// Process Simulation. All functionality packed into one method for easier overwriting
THIS^.Simulation();


// If enabled start station logic
IF THIS^.ipXtsSystem.Enabled THEN
	
	ipThisStation := (THIS^);
	//Detect mover who is passing the station whitout be in queue. Adjust to new Gap+Dynamics
	IF fbTrigger.MoverDetected AND fbTrigger.MoverAtTrigger<>0 AND NOT THIS^.bSuppressDynamicsChange THEN
		//Only if not in this queue
		IF fbTrigger.MoverAtTrigger.ParentStation <> ipThisStation THEN
			fbTrigger.MoverAtTrigger.MoveAbsCA(
				fPosition:= fbTrigger.MoverAtTrigger.LastCmdTargedPosition, 
				fVelocity:= THIS^.fMoverVelocityAtExit, 
				fGap:= THIS^.fMoverGapAtExit, 
				eDirection:= Tc3_Mc3Definitions.MC_DIRECTION.mcDirectionPositive);
		END_IF
	END_IF
	
	
	//Test if the first mover is in station and send him away, if the destination is not this station
	IF (THIS^.MoversInQueue[0] <> 0) AND_THEN (THIS^.MoversInQueue[0].TargedStation <> THIS^.StationGroupID) AND_THEN __QUERYINTERFACE(THIS^.MoversInQueue[0],ipMover) THEN
		//IF mover is standstill in current station, send him away whit the exitVelocity, else use the in mover stored velocity
		IF (THIS^.MoversInQueue[0].PositionOnTrack = THIS^.PositionOnTrack) THEN
			THIS^.TrySendMoverToNextStation(ipMover := ipMover, fVelocity := THIS^.fMoverVelocityAtExit, fGap := THIS^.fMoverGapAtExit);
		ELSE
			THIS^.TrySendMoverToNextStation(ipMover := ipMover, fVelocity := ipMover.LastCmdTargedVelocity, fGap := ipMover.LastCmdTargedGap);
		END_IF	
      
	END_IF
END_IF


// Utility InfoStation, used in XTS Viewer. All functionality packed into one method for easier overwriting
THIS^.UtilityStation();

// Calculate statistic values like Mover/min of this station. All functionality packed into one method for easier overwriting
THIS^.UpdateStatistic();
END_METHOD

METHOD PROTECTED UtilityStation : HRESULT //Utility InfoStation, used in XTS Viewer. All functionality packed into one method for easier overwriting
VAR
	aStopPositionsInfoStation : ARRAY[1..Tc3_XTS_Utility.TcIoXtsEnvironmentParameterList.MaxXtsStopPositionsPerStation] OF LREAL;
	fLastStopPosition 		: LREAL;
	nLoopIndex 				: UINT;	
    ipMovers 				: CHALET_BaseComponents.I_CH_List;
	ipTempMover 			: I_XTS_Mover;
	nXpuNo 					: UINT;
	nMoverNo 				: UINT;
END_VAR

VAR_INST
	bUtilityStationInitDone : BOOL;
	nOldMoverQueueSize 		: UINT := CHALET_BaseComponents.GVL_Datatypes.cMaxUint;
	fOldPositionOnTrack 	: LREAL;
	anBias 					: ARRAY[1..2] OF INT;
	bInverted 				: BOOL;
END_VAR
//Validate inputs
IF THIS^.OIDStationInfo = 0 OR ipXtsSystem.Environment = 0 THEN
	RETURN;
END_IF	


// Initalize
IF NOT bUtilityStationInitDone THEN
	//Get interface to utility station belongs to this station via OID
    FOR nLoopIndex := 1 TO ipXtsSystem.Environment.UtilityEnvirement.InfoServerTcIo(1).P_InfoStationCount DO
		IF 	ipXtsSystem.Environment.UtilityEnvirement.InfoServerTcIo(1).P_InfoStationOids[nLoopIndex] = THIS^.OIDStationInfo THEN
			THIS^.ipStationInfo := ipXtsSystem.Environment.UtilityEnvirement.InfoServerTcIo(1).InfoStationTcIo(nInfoStation:= nLoopIndex);
			EXIT;
		END_IF
	END_FOR	
	
	// calculate Position Offset
	IF THIS^.ipStationInfo <> 0 THEN			
		ipMovers := ipXtsSystem.Movers;
		ipMovers.ResetIterator();
		nLoopIndex := 0;	
		WHILE ipMovers.HasNextObject() DO
			nLoopIndex := nLoopIndex + 1;
			IF ToMover(ipMovers.GetNextObject(),ipTempMover) THEN
				//get Xpu Number by AxisId
				nXpuNo := ipXtsSystem.Environment.UtilityEnvirement.GetXpuNumberByAxisId(ipTempMover.getAxisRef.NcToPlc.AxisId);
				//get Mover Number by AxisId
				nMoverNo := ipXtsSystem.Environment.UtilityEnvirement.XpuTcIo(nXpuNo).GetMoverNumberByAxisId(ipTempMover.getAxisRef.NcToPlc.AxisId);
				//calculate Bias
				anBias[nLoopIndex] := LREAL_TO_INT(ipXtsSystem.Environment.UtilityEnvirement.XpuTcIo(nXpuNo).MoverTcIo(nMoverNo).GetPositionInfo().fPartPosition - ipTempMover.getAxisRef.NcToPlc.ModuloActPos);
				IF nLoopIndex = 2 THEN
					 EXIT;
				END_IF
			END_IF
		END_WHILE
		
		// Validate bias, check for inverted direction
		IF anBias[1] <> anBias[2] THEN
			bInverted := TRUE; 
			ipMovers.ResetIterator();
			nLoopIndex := 0;	
			WHILE ipMovers.HasNextObject() DO
				nLoopIndex := nLoopIndex + 1;
				IF ToMover(ipMovers.GetNextObject(),ipTempMover) THEN
					//get Xpu Number by AxisId
					nXpuNo := ipXtsSystem.Environment.UtilityEnvirement.GetXpuNumberByAxisId(ipTempMover.getAxisRef.NcToPlc.AxisId);
					//get Mover Number by AxisId
					nMoverNo := ipXtsSystem.Environment.UtilityEnvirement.XpuTcIo(nXpuNo).GetMoverNumberByAxisId(ipTempMover.getAxisRef.NcToPlc.AxisId);
					//calculate inverted Bias
					anBias[nLoopIndex] := LREAL_TO_INT(ipXtsSystem.TrackLength - ipXtsSystem.Environment.UtilityEnvirement.XpuTcIo(nXpuNo).MoverTcIo(nMoverNo).GetPositionInfo().fPartPosition - ipTempMover.getAxisRef.NcToPlc.ModuloActPos);
					IF nLoopIndex = 2 THEN
						 EXIT;
					END_IF
				END_IF	
			END_WHILE
		END_IF
		
		//Set unique station name
		THIS^.ipStationInfo.SetDescription(THIS^.LUID);

	END_IF
	bUtilityStationInitDone := TRUE;
END_IF




// Update
// Configure/draw station in viewer on change
IF (THIS^.ipStationInfo <> 0) AND (THIS^.nMoverQueueSize <> nOldMoverQueueSize OR THIS^.fPositionOnTrack <> fOldPositionOnTrack) THEN	
	nOldMoverQueueSize := THIS^.nMoverQueueSize;
	fOldPositionOnTrack := THIS^.fPositionOnTrack;
	
	
	
	// Draw stop position if gap between mover, given by station behind, is set
	IF (StationBehinde <> 0) AND (THIS^.nMoverQueueSize > 0) AND THIS^.nMoverQueueSize <= 25 THEN
		//Clear array
		MEMSET(ADR(aStopPositionsInfoStation), SIZEOF(aStopPositionsInfoStation), 0);
		//Fill array
		FOR nLoopIndex := 1 TO THIS^.nMoverQueueSize DO
			fLastStopPosition := (nLoopIndex-1)*StationBehinde.MoverGapAtExit;
			aStopPositionsInfoStation[(nLoopIndex)] := (fLastStopPosition);
		END_FOR
		IF NOT bInverted THEN
			//Start Position
			THIS^.ipStationInfo.SetStartPositionOnPart(MAX((fPositionOnTrack + anBias[1] - fLastStopPosition), 0)); ///zzz Todo. The InfoStation can not draw stations in the modulo area
			//End Pos
			THIS^.ipStationInfo.SetEndPositionOnPart(fPositionOnTrack + anBias[1]);
		ELSE
			//Start Position
			THIS^.ipStationInfo.SetStartPositionOnPart(ipXtsSystem.TrackLength - (fPositionOnTrack + anBias[1]));					
			//End Pos
			THIS^.ipStationInfo.SetEndPositionOnPart(MAX((ipXtsSystem.TrackLength - (fPositionOnTrack + anBias[1] - fLastStopPosition)), 0)); ///zzz Todo. The InfoStation can not draw stations in the modulo area
		END_IF
		//StopPositions
		THIS^.ipStationInfo.SetStopPositions(aStopPositionsInfoStation);

		//Override color if is set to transparent
		IF THIS^.ipStationInfo.GetStationColor() = 0 THEN
			THIS^.ipStationInfo.SetStationColor(nStationColor:= E_Colors_ARGB.Darkred);
		END_IF
	ELSE
		//Clear array
		MEMSET(ADR(aStopPositionsInfoStation), SIZEOF(aStopPositionsInfoStation), 0);	
		//StopPositions
		THIS^.ipStationInfo.SetStopPositions(aStopPositionsInfoStation);
		//Start Pos
		THIS^.ipStationInfo.SetStartPositionOnPart(nStartPositionOnPart := fPositionOnTrack + anBias[1]);
		//End Position
		THIS^.ipStationInfo.SetEndPositionOnPart(nEndPositionOnPart := fPositionOnTrack + anBias[1]);
	END_IF
	
	
	
	//Color Station depending on function:
	// Waitingstation green
	IF (FIND(THIS^.LUID,'wait')>0) OR (FIND(THIS^.LUID,'Wait')>0) OR (FIND(THIS^.LUID,'Warte')>0) OR (FIND(THIS^.LUID,'warte')>0) THEN
		THIS^.UtilityStationInfo.SetStationColor(nStationColor := E_Colors_ARGB.Green);
	
	// Dynamicstation blue
	ELSIF THIS^.MoverQueueSize = 0 THEN
		THIS^.UtilityStationInfo.SetStationColor(nStationColor := E_Colors_ARGB.Royalblue);	
    
	// Process station red
	ELSE
		THIS^.UtilityStationInfo.SetStationColor(nStationColor := E_Colors_ARGB.Red);			
	END_IF

END_IF
END_METHOD

{attribute 'monitoring':='call'}
PROPERTY UtilityStationInfo : I_TcIoXtsInfoServerInfoStation
GET
UtilityStationInfo := THIS^.ipStationInfo;
END_GET
END_PROPERTY

END_FUNCTION_BLOCK

// COMPENENTs/Trigger/FB_XTS_Trigger
{attribute 'no_explicit_call' := 'Do not call the body - Stick to OOP'}
FUNCTION_BLOCK FB_XTS_Trigger EXTENDS FB_CH_Object IMPLEMENTS I_XTS_Trigger
VAR
	{attribute 'hide'}
	bInitDone : BOOL;
	{attribute 'hide'}
	ipXtsSystem : I_XTS_System_Registration;
	{attribute 'hide'}
	ipListOfMoversToCheck : CHALET_BaseComponents.I_CH_LIST;
	{attribute 'hide'}
	fTriggerPositionOnTrack : LREAL;
	{attribute 'hide'}
	eTriggerDirection : Tc2_MC2.MC_Direction := MC_Positive_Direction;
	{attribute 'hide'}
	ipMoverAtTrigger : I_XTS_Mover;
	{attribute 'hide'}	
	fTrackLentgh : LREAL;
	{attribute 'hide'}
	aMoversPositionLastCycle : ARRAY [0..(XtsParameterlist.MAX_MOVER_PER_SYSTEM-1)] OF LREAL; // This list is generated at the end of the PRG and contais the positions. The positions are checked in the next cycle
	{attribute 'hide'}
	aMoversInterfaceLastCycle : ARRAY [0..(XtsParameterlist.MAX_MOVER_PER_SYSTEM-1)] OF I_XTS_Mover; // This list is generated at the end of the PRG and contais the Mover interface. The positions are checked in the next cycle
	
END_VAR

METHOD FB_init : BOOL
VAR_INPUT
	bInitRetains : BOOL; // if TRUE, the retain variables are initialized (warm start / cold start)
	bInCopyCode : BOOL;  // if TRUE, the instance afterwards gets moved into the copy code (online change)
	
	ipXtsSystem : I_XTS_System_Registration; //Interface to XTS system object
	
END_VAR
VAR_INST
	{attribute 'hide'}
	bFBInitCalledOnce : BOOL; //Do the following code once during start up and not during onlinechange
END_VAR
//Do the following code once during start up and not during onlinechange
IF NOT bFBInitCalledOnce THEN 
	;
END_IF

//Regristrate object in System if unknown
IF ipXtsSystem <> 0 AND THIS^.ipXtsSystem = 0 THEN
	ipXtsSystem.RegisterTrigger(THIS^);
	THIS^.ipXtsSystem := ipXtsSystem;
END_IF

bFBInitCalledOnce := TRUE;
END_METHOD

{attribute 'monitoring':='call'}
PROPERTY HR : HRESULT
GET
///zzz todo
END_GET
END_PROPERTY

METHOD Initialize : HRESULT
IF THIS^.ipXtsSystem = 0 THEN
	//No valide interface
	Initialize := E_FAIL;
	RETURN;
END_IF

//Store track information
THIS^.fTrackLentgh := THIS^.ipXtsSystem.TrackLength;

IF (THIS^.ipListOfMoversToCheck <> 0) AND (THIS^.fTrackLentgh > 0.0) THEN
	THIS^.bInitDone := TRUE;
	Initialize := S_OK;
ELSE
	Initialize := E_FAIL;
END_IF
END_METHOD

PROPERTY ListOfMoversToCheck : I_CH_List
SET
IF ListOfMoversToCheck <> 0 THEN
	ipListOfMoversToCheck := ListOfMoversToCheck;
END_IF
END_SET
END_PROPERTY

{attribute 'monitoring':='call'}
PROPERTY MoverAtTrigger : I_XTS_Mover
GET
THIS^.Prepare();//Prepare Time-critical information

MoverAtTrigger := ipMoverAtTrigger;
END_GET
END_PROPERTY

{attribute 'monitoring':='call'}
PROPERTY MoverDetected : BOOL
GET
THIS^.Prepare();//Prepare Time-critical information

MoverDetected := (ipMoverAtTrigger <> 0);
END_GET
END_PROPERTY

{attribute 'monitoring':='call'}
PROPERTY PositionOnTrack : LREAL
GET
PositionOnTrack := fTriggerPositionOnTrack;
END_GET
SET
fTriggerPositionOnTrack := PositionOnTrack;
END_SET
END_PROPERTY

(* Time-critical information is processed here, which can then be polled via the property every cycle. 
The update method is usually at the end of the program and then it is already 'outdated'. *)
METHOD PRIVATE Prepare : HRESULT
VAR
	fMoverActPos,fMoverLastPos : LREAL;
	fRangePositive, fRangeNegative : LREAL;
	bMoverWasInRangeNeg, bMoverWasInRangePos, bMoverIsInRangeNeg, bMoverIsInRangePos : BOOL;
	nLoopIndex : UINT;
END_VAR
VAR_INST
	{attribute 'hide'}
	nLastUpdatedCycleCount : UDINT;
END_VAR
VAR CONSTANT
	cMaxMoveDistPerCycle : LREAL := 4000.0 * 20.0 / 1000.0 * 1.1; //4 m/s(max. XTS speed) * 20ms(max realistic SPS cycle time) + 10%
END_VAR
//Check if this Cycle the dates are allready prepared
IF nLastUpdatedCycleCount <> TwinCAT_SystemInfoVarList._TaskInfo[THIS^.nTaskIndex].CycleCount THEN
	nLastUpdatedCycleCount := TwinCAT_SystemInfoVarList._TaskInfo[THIS^.nTaskIndex].CycleCount;

	//Clear last stored Mover if an new cycle has started
	THIS^.ipMoverAtTrigger := 0;
	
	//Check old list of Moverspositions and compare them to the current position of the same mover.
	//Set Trigger if the Mover pass the Station
	fRangePositive := LMOD(lr_Value:=(THIS^.fTriggerPositionOnTrack + cMaxMoveDistPerCycle + THIS^.fTrackLentgh),lr_Arg:= THIS^.fTrackLentgh);
	fRangeNegative := LMOD(lr_Value:=(THIS^.fTriggerPositionOnTrack - cMaxMoveDistPerCycle + THIS^.fTrackLentgh),lr_Arg:= THIS^.fTrackLentgh);
	
	FOR nLoopIndex := 0 TO (XtsParameterlist.MAX_MOVER_PER_SYSTEM-1) DO
		IF aMoversInterfaceLastCycle[nLoopIndex] <> 0 THEN
			fMoverActPos :=  aMoversInterfaceLastCycle[nLoopIndex].PositionOnTrack;
			fMoverLastPos:=  aMoversPositionLastCycle[nLoopIndex];
			
			
			//Test if the the Mover was in Trigger-100mm Range(without exact the trigger point) and is now in Trigger+100 Range(with exact the trigger point)
			bMoverWasInRangePos	:= FUN_InLimitTest(fMinimum :=THIS^.fTriggerPositionOnTrack, fInput:= fMoverLastPos, fMaximum:=fRangePositive) AND NOT (fMoverLastPos=THIS^.fTriggerPositionOnTrack); 
			bMoverWasInRangeNeg	:= FUN_InLimitTest(fMinimum :=fRangeNegative, fInput:= fMoverLastPos, fMaximum:=THIS^.fTriggerPositionOnTrack) AND NOT (fMoverLastPos=THIS^.fTriggerPositionOnTrack); 
			bMoverIsInRangePos 	:= FUN_InLimitTest(fMinimum :=THIS^.fTriggerPositionOnTrack, fInput:= fMoverActPos, fMaximum:=fRangePositive); 
			bMoverIsInRangeNeg 	:= FUN_InLimitTest(fMinimum :=fRangeNegative, fInput:= fMoverActPos, fMaximum:=THIS^.fTriggerPositionOnTrack); 
		
			IF eTriggerDirection = MC_Positive_Direction AND bMoverWasInRangeNeg AND bMoverIsInRangePos THEN
				THIS^.ipMoverAtTrigger := aMoversInterfaceLastCycle[nLoopIndex];
				RETURN;
			ELSIF eTriggerDirection = MC_Negative_Direction AND bMoverIsInRangeNeg AND bMoverWasInRangePos THEN
				THIS^.ipMoverAtTrigger := aMoversInterfaceLastCycle[nLoopIndex];
				RETURN;	
			END_IF
			
		END_IF
	END_FOR
END_IF
END_METHOD

{attribute 'monitoring':='call'}
PROPERTY TimeStamp : Tc2_EtherCAT.T_DCTIME64
GET
THIS^.Prepare();//Prepare Time-critical information

///zzz todo exact time stamp calculatioin
 IF ipMoverAtTrigger <> 0 THEN
	 TimeStamp := F_GetCurDcTaskTime64();
 ELSE
	 TimeStamp := 0;
 END_IF
END_GET
END_PROPERTY

{attribute 'monitoring':='call'}
PROPERTY TriggerDirection : Tc2_MC2.MC_Direction
GET
TriggerDirection := eTriggerDirection;
END_GET
SET
IF TriggerDirection = MC_Positive_Direction OR TriggerDirection = MC_Negative_Direction THEN
	eTriggerDirection := TriggerDirection;
END_IF
END_SET
END_PROPERTY

METHOD Update : HRESULT
VAR
	nIndex : UINT;
	ipMover : I_XTS_Mover;
END_VAR
//Force to do an init befor call update
IF NOT bInitDone THEN
	THIS^.Initialize();
	RETURN;
END_IF

//Clear array
MEMSET(destAddr:=ADR(aMoversInterfaceLastCycle),n:=SIZEOF(aMoversInterfaceLastCycle),fillByte:=0);
MEMSET(destAddr:=ADR(aMoversPositionLastCycle),n:=SIZEOF(aMoversPositionLastCycle),fillByte:=0);

nIndex := 0;
THIS^.ipListOfMoversToCheck.ResetIterator();
WHILE THIS^.ipListOfMoversToCheck.HasNextObject() DO
	
	//Cheack all Movers fill the actposition in the array
	IF ToMover(THIS^.ipListOfMoversToCheck.GetNextObject(),ipMover) THEN
		aMoversInterfaceLastCycle[nIndex] := ipMover;
		aMoversPositionLastCycle[nIndex] := ipMover.PositionOnTrack;
		nIndex := nIndex +1;
	END_IF
	
END_WHILE
END_METHOD

END_FUNCTION_BLOCK

// FUNCTIONs/FUN_InLimitTest
FUNCTION FUN_InLimitTest : BOOL
VAR_INPUT
	fMinimum 	: LREAL;
	fMaximum 	: LREAL;
	fInput 		: LREAL;
END_VAR

//Normal case
// 9 Max
// 5 Test
// 1 Min
IF fMinimum <= fMaximum THEN
	FUN_InLimitTest := (fInput >= fMinimum) AND (fInput <= fMaximum);
	
//Modulo case	
// 6 | 6  Max
// 5 | 9  Test
// 8 | 8  Min
ELSIF fMinimum > fMaximum THEN
	FUN_InLimitTest := NOT((fInput > fMaximum) AND (fInput < fMinimum));
END_IF

END_FUNCTION

// COMPENENTs/Zone/FB_XTS_Zone
{attribute 'no_explicit_call' := 'Do not call the body - Stick to OOP'}
// Check zone start to end in positive direktion.
FUNCTION_BLOCK FB_XTS_Zone EXTENDS FB_CH_Object IMPLEMENTS I_XTS_Zone
VAR
	{attribute 'hide'}
	bInitDone : BOOL;
	{attribute 'hide'}
	ipXtsSystem : I_XTS_System_Registration;
	
	{attribute 'hide'}
	ipListOfMoversToCheck : CHALET_BaseComponents.I_CH_LIST;
	{attribute 'hide'}
	aMoversInZone : ARRAY [0..(XtsParameterlist.MAX_MOVER_PER_SYSTEM-1)] OF I_XTS_Mover_PLC;
	{attribute 'hide'}
	fStartPositionOnTrack : LREAL;
	{attribute 'hide'}
	fEndPositionOnTrack : LREAL;	
	{attribute 'hide'}
	fTrackLentgh : LREAL;
END_VAR

{attribute 'monitoring':='call'}
PROPERTY CtsMoversInZone : UINT
GET
VAR
	nIndex : UINT;
END_VAR
THIS^.Prepare();//Prepare Time-critical information

//Check array for entrys, exit if fisrt empty arrayindex is found.
FOR nIndex := 0 TO (XtsParameterlist.MAX_MOVER_PER_SYSTEM-1) DO
	IF (aMoversInZone[nIndex] <> 0) THEN
		CtsMoversInZone := CtsMoversInZone +1;
	ELSE
		RETURN;
	END_IF
END_FOR
END_GET
END_PROPERTY

{attribute 'monitoring':='call'}
PROPERTY EndPositionOnTrack : LREAL
GET
EndPositionOnTrack := fEndPositionOnTrack;
END_GET
SET
fEndPositionOnTrack := EndPositionOnTrack;
END_SET
END_PROPERTY

METHOD FB_init : BOOL
VAR_INPUT
	bInitRetains : BOOL; // if TRUE, the retain variables are initialized (warm start / cold start)
	bInCopyCode : BOOL;  // if TRUE, the instance afterwards gets moved into the copy code (online change)
	
	ipXtsSystem : I_XTS_System_Registration; //Interface to XTS system object
END_VAR
VAR_INST
	{attribute 'hide'}
	bFBInitCalledOnce : BOOL; //Do the following code once during start up and not during onlinechange
END_VAR
//Do the following code once during start up and not during onlinechange
IF NOT bFBInitCalledOnce THEN 
	;
END_IF

//Regristrate object in System if unknown
IF ipXtsSystem <> 0 AND THIS^.ipXtsSystem = 0 THEN
	ipXtsSystem.RegisterZone(THIS^);
	THIS^.ipXtsSystem := ipXtsSystem;
END_IF

bFBInitCalledOnce := TRUE;
END_METHOD

{attribute 'monitoring':='call'}
PROPERTY HR : HRESULT
GET
IF CHALET_BaseComponents.BaseParameterlist.MAX_OBJECTS > XtsParameterlist.MAX_MOVER_PER_SYSTEM THEN
	HR := E_FAIL;
END_IF
END_GET
END_PROPERTY

METHOD Initialize : HRESULT
IF THIS^.ipXtsSystem = 0 THEN
	//No valide interface
	Initialize := E_FAIL;
	RETURN;
END_IF

//Store track information
THIS^.fTrackLentgh := THIS^.ipXtsSystem.TrackLength;

IF (THIS^.ipListOfMoversToCheck <> 0) AND (THIS^.fTrackLentgh > 0.0) THEN
	THIS^.bInitDone := TRUE;
	Initialize := S_OK;
ELSE
	Initialize := E_FAIL;
END_IF
END_METHOD

PROPERTY ListOfMoversToCheck : I_CH_List
SET
IF ListOfMoversToCheck <> 0 THEN
	ipListOfMoversToCheck := ListOfMoversToCheck;
END_IF
END_SET
END_PROPERTY

{attribute 'monitoring':='call'}
PROPERTY MoversInZone : REFERENCE TO ARRAY [0..(XtsParameterlist.MAX_MOVER_PER_SYSTEM-1)] OF I_XTS_Mover_PLC // Return a sorted list of movers in this zone. Index 0 is the mover in Front.
GET
THIS^.Prepare();//Prepare Time-critical information

MoversInZone REF= THIS^.aMoversInZone;
END_GET
END_PROPERTY

(* Time-critical information is processed here, which can then be polled via the property every cycle. 
The update method is usually at the end of the program and then it is already 'outdated'. *)
METHOD PRIVATE Prepare : HRESULT
VAR
	nLoopIndex : UINT;
	ipMoverPlc : I_XTS_Mover_PLC;
	fDistToStart : LREAL;
	aDisanceToStart : ARRAY [0..XtsParameterlist.MAX_MOVER_PER_SYSTEM] OF LREAL;
END_VAR
VAR_INST
	{attribute 'hide'}
	nLastUpdatedCycleCount : UDINT;
END_VAR
//Check if this Cycle the dates are allready prepared
IF nLastUpdatedCycleCount <> TwinCAT_SystemInfoVarList._TaskInfo[THIS^.nTaskIndex].CycleCount THEN
	nLastUpdatedCycleCount := TwinCAT_SystemInfoVarList._TaskInfo[THIS^.nTaskIndex].CycleCount;

	//Clear array
	MEMSET(destAddr:=ADR(aMoversInZone),n:=SIZEOF(aMoversInZone),fillByte:=0);
	
	//Cheack all Movers and generate a sorted list of all mover in this zone
	THIS^.ipListOfMoversToCheck.ResetIterator();
	WHILE THIS^.ipListOfMoversToCheck.HasNextObject() DO
		IF ToMover_PLC(THIS^.ipListOfMoversToCheck.GetNextObject(),ipMoverPlc) THEN
			
			//If in zone
			IF FUN_InLimitTest(fMinimum:= fStartPositionOnTrack, fMaximum:=fEndPositionOnTrack, fInput:= ipMoverPlc.PositionOnTrack) THEN
				fDistToStart := FUN_GetDistToPosModulo(fActualPosition:= ipMoverPlc.PositionOnTrack, fTargedPosition:= fEndPositionOnTrack, fModulo := fTrackLentgh);
				
				//Check array of movers and decide if the current one is closer to 
				FOR nLoopIndex := 0 TO (XtsParameterlist.MAX_MOVER_PER_SYSTEM-1) DO
					//empty array position
					IF aMoversInZone[nLoopIndex] = 0 THEN
						aMoversInZone[nLoopIndex] := ipMoverPlc;
						aDisanceToStart[nLoopIndex] := fDistToStart;
						EXIT;
						
					//Closer Mover found, move whole array 	
					ELSIF aDisanceToStart[nLoopIndex] > fDistToStart THEN
						MEMMOVE(srcAddr := ADR(aMoversInZone[nLoopIndex]), destAddr := ADR(aMoversInZone[nLoopIndex+1]), n := (SIZEOF(aMoversInZone[0])*(XtsParameterlist.MAX_MOVER_PER_SYSTEM-nLoopIndex-1)));
						MEMMOVE(srcAddr := ADR(aDisanceToStart[nLoopIndex]), destAddr := ADR(aDisanceToStart[nLoopIndex+1]), n := (SIZEOF(aDisanceToStart[0])*(XtsParameterlist.MAX_MOVER_PER_SYSTEM-nLoopIndex-1)));
						aMoversInZone[nLoopIndex] := ipMoverPlc;
						aDisanceToStart[nLoopIndex] := fDistToStart;
						EXIT;
						
					//check next position	
					ELSE 
						;
					END_IF
				END_FOR
			END_IF
		END_IF
	END_WHILE
END_IF
END_METHOD

{attribute 'monitoring':='call'}
PROPERTY StartPositionOnTrack : LREAL
GET
StartPositionOnTrack := fStartPositionOnTrack;
END_GET
SET
fStartPositionOnTrack := StartPositionOnTrack;
END_SET
END_PROPERTY

METHOD Update : HRESULT
VAR

END_VAR
// Nothing todo in Update. Check Prepare
END_METHOD

END_FUNCTION_BLOCK

// COMPENENTs/Zone/I_XTS_Zone
INTERFACE I_XTS_Zone

{attribute 'monitoring':='call'}
PROPERTY CtsMoversInZone : UINT
GET
END_GET
END_PROPERTY

{attribute 'monitoring':='call'}
PROPERTY EndPositionOnTrack : LREAL
GET
END_GET
SET
END_SET
END_PROPERTY

{attribute 'monitoring':='call'}
PROPERTY HR : HRESULT
GET
END_GET
END_PROPERTY

PROPERTY ListOfMoversToCheck : I_CH_List
SET
END_SET
END_PROPERTY

{attribute 'monitoring':='call'}
PROPERTY MoversInZone : REFERENCE TO ARRAY [0..(XtsParameterlist.MAX_MOVER_PER_SYSTEM-1)] OF I_XTS_Mover_PLC
GET
END_GET
END_PROPERTY

{attribute 'monitoring':='call'}
PROPERTY StartPositionOnTrack : LREAL
GET
END_GET
SET
END_SET
END_PROPERTY

END_INTERFACE

// FUNCTIONs/FUN_GetDistToPosModulo
FUNCTION FUN_GetDistToPosModulo : LREAL //This is only working in Positiv Direktion
VAR_INPUT
	fTargedPosition : LREAL;
	fActualPosition : LREAL;
	fModulo 		: LREAL;
END_VAR

VAR

END_VAR

IF fTargedPosition < fActualPosition THEN
	fTargedPosition := fTargedPosition + fModulo;
END_IF

FUN_GetDistToPosModulo := fTargedPosition - fActualPosition;

END_FUNCTION

// FUNCTIONs/FUN_BuildLogString
FUNCTION FUN_BuildLogString : String
VAR_INPUT
	fPos : LREAL;
	fVelocity : LREAL;
	fGap : LREAL;
END_VAR
VAR
	sTemp: STRING;
END_VAR

sTemp := 				CONCAT('Pos:' , LREAL_TO_STRING(fPos));
sTemp := CONCAT(sTemp, 	CONCAT(', Velocity:' , LREAL_TO_STRING(fVelocity)));
sTemp := CONCAT(sTemp, 	CONCAT(', Gap:' , LREAL_TO_STRING(fGap)));

FUN_BuildLogString := sTemp;

END_FUNCTION

// COMPENENTs/System/FB_XTS_System
{attribute 'no_explicit_call' := 'Do not call the body - Stick to OOP'}
FUNCTION_BLOCK FB_XTS_System EXTENDS FB_CH_Object IMPLEMENTS I_XTS_System_Registration, I_XTS_System_PLC
VAR	
	{attribute 'hide'}
	bInitDone : BOOL;
	bErrorDuringFbInit : BOOL; // Not possible to reset
	{attribute 'hide'}
    fbMovers     : CHALET_BaseComponents.FB_CH_List;
	{attribute 'hide'}	
	fbStations 	 : CHALET_BaseComponents.FB_CH_List;
	{attribute 'hide'}	
	fbZones 	 : CHALET_BaseComponents.FB_CH_List;
	{attribute 'hide'}	
	fbTriggers 	 : CHALET_BaseComponents.FB_CH_List;
	{attribute 'hide'}	
	ipGroup		 : I_XTS_Group;
	{attribute 'hide'}	
    ipEnvironment : I_XTS_Environment;
	{attribute 'hide'}
    nState_SEQ_Enabling  : UINT;
	{attribute 'hide'}	
    nState_SEQ_Disabling  : UINT;
	{attribute 'hide'}	
	fbFeedback : CHALET_BaseComponents.FB_CH_Feedback;
END_VAR

METHOD Disable : CHALET_BaseComponents.I_CH_Feedback
//Disable is allways posible

THIS^.nState_SEQ_Disabling 	:= 1;
THIS^.nState_SEQ_Enabling 	:= 0;

//prevent a mover from a station from getting a new position at high speed when stopped
THIS^.SuppressAllDynamicsChanges := TRUE;	

THIS^.fbFeedback.LastCommandAccepted:= TRUE;
THIS^.fbFeedback.ActiveCommand 		:= 'Disable';
THIS^.fbFeedback.Busy 				:= TRUE;	
Disable := THIS^.fbFeedback;
END_METHOD

{attribute 'monitoring':='call'}
PROPERTY Disabled : BOOL
GET
Disabled := nState_SEQ_Disabling = 999 OR 
			(nState_SEQ_Disabling = 0 AND nState_SEQ_Enabling = 0);
END_GET
END_PROPERTY

METHOD PROTECTED Disabling : HRESULT
VAR
	hr : HRESULT;
	bOk : BOOL := TRUE;
	ipTempMover : I_XTS_Mover;
END_VAR

VAR_INST
	fbTimeWait : TON; 
	hrLastCycle : HRESULT;
END_VAR
Disabling := S_PENDING;
CASE nState_SEQ_Disabling OF
	0: // Idle
		Disabling := S_OK;
		
		
	1: // Halt movers
		THIS^.fbMovers.ResetIterator();
		WHILE THIS^.fbMovers.HasNextObject() DO
			IF ToMover(THIS^.fbMovers.GetNextObject(),ipTempMover) THEN
				IF ipTempMover.MoverInGroup AND NOT ipTempMover.getAxisRef.Status.HasBeenStopped THEN
					hr := GetMostSignificant(hr, ipTempMover.HaltCA());
				END_IF
			END_IF
		END_WHILE
		
		//Ignore feedback at this step. in next seq the movers get reseted.
		nState_SEQ_Disabling := 20;
		
	20: // Halting movers	
		THIS^.fbMovers.ResetIterator();
		WHILE THIS^.fbMovers.HasNextObject() DO
			IF ToMover(THIS^.fbMovers.GetNextObject(),ipTempMover) THEN
				bOk := bOk AND ipTempMover.getAxisRef.NcToPlc.SetVelo = 0;
			END_IF
		END_WHILE
		
		IF bOk THEN 
			nState_SEQ_Disabling := 25;
		END_IF	
		
		
	25: // wait for halt done
		IF THIS^.ipGroup.AllAxesStanding THEN
			nState_SEQ_Disabling := 30;
		END_IF
					
		
	30: // Reset movers
		THIS^.fbMovers.ResetIterator();
		WHILE THIS^.fbMovers.HasNextObject() DO
			IF ToMover(THIS^.fbMovers.GetNextObject(),ipTempMover) THEN
				hr := GetMostSignificant(hr, ipTempMover.Reset());
			END_IF
		END_WHILE
		
		IF CheckOk(hr) THEN 
			nState_SEQ_Disabling := 40;
		ELSE
			nState_SEQ_Disabling := 1000 + nState_SEQ_Disabling;
		END_IF				
		
		
	40: // Resetting movers
		THIS^.fbMovers.ResetIterator();
		WHILE THIS^.fbMovers.HasNextObject() DO
			IF ToMover(THIS^.fbMovers.GetNextObject(),ipTempMover) THEN
				hr := GetMostSignificant(hr, ipTempMover.Feedback.HR);
			END_IF
		END_WHILE
		
		IF CheckOk(hr) THEN 
			nState_SEQ_Disabling := 63;
		ELSIF FAILED(hr) THEN
			nState_SEQ_Disabling := 1000 + nState_SEQ_Disabling;
		END_IF
	
		
	63: // Reset group
		hr :=  THIS^.ipGroup.Reset();
		
		IF CheckOk(hr) THEN 
			nState_SEQ_Disabling := 64;
		ELSE
			nState_SEQ_Disabling := 1000 + nState_SEQ_Disabling;
		END_IF		
		
		
	64: // Resetting group
		hr := THIS^.ipGroup.HR;
		
		IF CheckOk(hr) THEN 
			nState_SEQ_Disabling := 70;
		ELSIF FAILED(hr) THEN
			nState_SEQ_Disabling := 1000 + nState_SEQ_Disabling;
		END_IF		
		
		
	70: // Disable group
		hr := THIS^.ipGroup.Disable();
		
		IF CheckOk(hr) THEN 
			nState_SEQ_Disabling := 100;
		ELSE
			nState_SEQ_Disabling := 1000 + nState_SEQ_Disabling;
		END_IF	
		
		
   100: // Disabling group
		hr := THIS^.ipGroup.HR;
		
		IF CheckOk(hr) THEN 
			nState_SEQ_Disabling := 110;
		ELSIF FAILED(hr) THEN
			nState_SEQ_Disabling := 1000 + nState_SEQ_Disabling;
		END_IF			
		
		
	110: // Remove movers from group
		hr := THIS^.ipGroup.UngroupAllAxes();
		
		IF CheckOk(hr) THEN 
			nState_SEQ_Disabling := 120;
		ELSE
			nState_SEQ_Disabling := 1000 + nState_SEQ_Disabling;
		END_IF		
	
		
	120: // Removing movers from group
		hr := THIS^.ipGroup.HR;
		
		IF CheckOk(hr) THEN 
			nState_SEQ_Disabling := 130;
		ELSIF FAILED(hr) THEN
			nState_SEQ_Disabling := 1000 + nState_SEQ_Disabling;
		END_IF	

		
	130: // write state to movers
		THIS^.fbMovers.ResetIterator();
		WHILE THIS^.fbMovers.HasNextObject() DO
			IF ToMover(THIS^.fbMovers.GetNextObject(),ipTempMover) THEN
				ipTempMover.MoverInGroup := FALSE;
			END_IF
		END_WHILE

		nState_SEQ_Disabling := 170;	
		
		
	170: // Disable movers
		THIS^.fbMovers.ResetIterator();
		WHILE THIS^.fbMovers.HasNextObject() DO
			IF ToMover(THIS^.fbMovers.GetNextObject(),ipTempMover) THEN
				hr := GetMostSignificant(hr, ipTempMover.Disable());
			END_IF
		END_WHILE
		
		IF CheckOk(hr) THEN 
			nState_SEQ_Disabling := 180;
		ELSE
			nState_SEQ_Disabling := 1000 + nState_SEQ_Disabling;
		END_IF			
		
		
	180: // Disabling movers
		THIS^.fbMovers.ResetIterator();
		WHILE THIS^.fbMovers.HasNextObject() DO
			IF ToMover(THIS^.fbMovers.GetNextObject(),ipTempMover) THEN
				hr := GetMostSignificant(hr, ipTempMover.Feedback.HR);
			END_IF
		END_WHILE
		
		IF CheckOk(hr) THEN 
			nState_SEQ_Disabling := 200;
		ELSIF FAILED(hr) THEN
			nState_SEQ_Disabling := 1000 + nState_SEQ_Disabling;
		END_IF		

		
	200: // Wait 1 second according to documentation
		fbTimeWait.IN := TRUE;
		fbTimeWait.PT := T#1S;	
		fbTimeWait();
		
		IF fbTimeWait.Q THEN
			fbTimeWait.IN := FALSE;
			fbTimeWait();
			nState_SEQ_Disabling := 999;
		END_IF
	
		
   999: //Done
   		Disabling := S_OK;

		
	1000..1999://Error
		hr := GetMostSignificant(hrLastCycle, E_FAIL);	
END_CASE


//store last information
hrLastCycle := hr;


// Propagate error
IF FAILED(hr) THEN
	Disabling := hr;
END_IF
END_METHOD

METHOD Enable : CHALET_BaseComponents.I_CH_Feedback
IF NOT THIS^.fbFeedback.Done THEN
	//Error active/not ready
	THIS^.fbFeedback.LastCommandAccepted 	:= FALSE;

ELSIF nState_SEQ_Enabling <> 0 THEN
	//System is partial or full enabled. Disable first.
	THIS^.fbFeedback.LastCommandAccepted 	:= FALSE;
ELSE
	
	THIS^.SuppressAllDynamicsChanges := FALSE;	

	THIS^.nState_SEQ_Disabling 	:= 0;
	THIS^.nState_SEQ_Enabling 	:= 1;
	THIS^.fbFeedback.LastCommandAccepted 	:= TRUE;
	THIS^.fbFeedback.ActiveCommand 			:= 'Enable';
	THIS^.fbFeedback.Busy 				 	:= TRUE;	
END_IF

Enable := THIS^.fbFeedback;
END_METHOD

{attribute 'monitoring':='call'}
PROPERTY Enabled : BOOL
GET
Enabled := nState_SEQ_Enabling = 999;
END_GET
END_PROPERTY

METHOD PROTECTED Enabling : HRESULT
VAR
	hr : HRESULT;

	ipTempMover 	: I_XTS_Mover;
END_VAR

VAR_INST
	fbTimeOutSeq 	: TON; 
	hrLastCycle 	: HRESULT;
	nModuleCount 	: UDINT;
	nLoopCount 		: UDINT;
END_VAR
Enabling := S_PENDING;
CASE nState_SEQ_Enabling OF
	0: // Idle
		Enabling := S_OK;

	1: // Check OP mode
		IF THIS^.ipEnvironment.UtilityEnvirement.XpuTcIo(1).GetOperationMode() = OperationMode.Normal THEN
			nState_SEQ_Enabling := 2; // Check 48V of all Module
		ELSE
			nState_SEQ_Enabling := 3; // in Simulation check of 48V not necessary
		END_IF
		
		
	2: // ToDo: check 48V of all Module?
		nModuleCount:= THIS^.ipEnvironment.UtilityEnvirement.XpuTcIo(1).PartTcIo(1).GetModuleCount();
		nState_SEQ_Enabling := 3;
		FOR nLoopCount := 1 TO nModuleCount DO
			IF THIS^.ipEnvironment.UtilityEnvirement.XpuTcIo(1).PartTcIo(1).ModuleTcIo(UDINT_TO_UINT(nLoopCount)).GetDCLinkVoltage() < 20 AND
			   THIS^.ipEnvironment.UtilityEnvirement.XpuTcIo(1).PartTcIo(1).ModuleTcIo(UDINT_TO_UINT(nLoopCount)).GetDCLinkVoltage() > 56 THEN	
				nState_SEQ_Enabling := 2;				     
			END_IF		
		END_FOR

		
	3: // ask for MoverId Detection Mode	
		IF Environment.UtilityEnvirement.XpuTcIo(1).GetMoverIdDetectionMode() = MoverIdDetectionMode.Standard THEN			
			nState_SEQ_Enabling := 10;
		ELSIF Environment.UtilityEnvirement.XpuTcIo(1).GetMoverIdDetectionMode() = MoverIdDetectionMode.Mover1 THEN
			nState_SEQ_Enabling := 5;
		ELSE // todo: MoverIdDetectionMode.MultipleMover1
			;
		END_IF
		

	5: // Trigger Mover ID dedection 
		IF NOT Environment.UtilityEnvirement.XpuTcIo(1).GetIsMoverIdDetectionActive() AND
		   NOT Environment.UtilityEnvirement.XpuTcIo(1).GetIsMoverIdDetectionValid() THEN
			// Set the Trigger for ID detection
			Environment.UtilityEnvirement.XpuTcIo(1).TriggerMoverIdDetection();
		ELSIF Environment.UtilityEnvirement.XpuTcIo(1).GetIsMoverIdDetectionValid() THEN
			// successful
			nState_SEQ_Enabling := 10;
		ELSIF Environment.UtilityEnvirement.XpuTcIo(1).GetHasMoverIdDetectionError() THEN
			// error
			nState_SEQ_Enabling := 1000 + nState_SEQ_Enabling;
		ELSE 
			; // wait for valid or error					
		END_IF
		
	
	10: // Reset movers
		THIS^.fbMovers.ResetIterator();
		WHILE THIS^.fbMovers.HasNextObject() DO
			IF ToMover(THIS^.fbMovers.GetNextObject(), ipTempMover) THEN
				hr := GetMostSignificant(hr, ipTempMover.Reset());
			END_IF
		END_WHILE
		
		IF CheckOk(hr) THEN 
			nState_SEQ_Enabling := 20;
		ELSE
			nState_SEQ_Enabling := 1000 + nState_SEQ_Enabling;
		END_IF
		
		
	20: // Resetting movers
		THIS^.fbMovers.ResetIterator();
		WHILE THIS^.fbMovers.HasNextObject() DO
			IF toMover(THIS^.fbMovers.GetNextObject(), ipTempMover) THEN
				hr := GetMostSignificant(hr, ipTempMover.Feedback.HR);
			END_IF
		END_WHILE
		
		IF CheckOk(hr) THEN 
			nState_SEQ_Enabling := 110;
		ELSIF FAILED(hr) THEN
			nState_SEQ_Enabling := 1000 + nState_SEQ_Enabling;
		END_IF	

	102: // ToDo: Config Station?
	
	103: // ToDo: Configuring Stations?
	
	
	110: // Enable movers
		THIS^.fbMovers.ResetIterator();
		WHILE THIS^.fbMovers.HasNextObject() DO
			IF ToMover(THIS^.fbMovers.GetNextObject(),ipTempMover) THEN
				hr := GetMostSignificant(hr, ipTempMover.Enable());				 
			END_IF
		END_WHILE
		
		IF CheckOk(hr) THEN 
			nState_SEQ_Enabling := 120;
		ELSE
			nState_SEQ_Enabling := 1000 + nState_SEQ_Enabling;
		END_IF	
		

	120: // Enabling movers
		THIS^.fbMovers.ResetIterator();
		WHILE THIS^.fbMovers.HasNextObject() DO
			IF ToMover(THIS^.fbMovers.GetNextObject(),ipTempMover) THEN
				hr := GetMostSignificant(hr, ipTempMover.Feedback.HR);	
			END_IF
		END_WHILE
		
		IF CheckOk(hr) THEN 
			nState_SEQ_Enabling := 130;
		ELSIF FAILED(hr) THEN
			nState_SEQ_Enabling := 1000 + nState_SEQ_Enabling;
		END_IF
		
		
	130: // Add movers to group
		hr := THIS^.ipGroup.AddAxisListToGroup(fbMovers);
		
		IF CheckOk(hr) THEN 
			nState_SEQ_Enabling := 140;
		ELSE
			nState_SEQ_Enabling := 1000 + nState_SEQ_Enabling;
		END_IF	
		

	140: // Adding mover to group
		hr := THIS^.ipGroup.AddingAxisToGroup();
		
		IF CheckOk(hr) THEN 
			nState_SEQ_Enabling := 150;
		ELSIF FAILED(hr) THEN
			nState_SEQ_Enabling := 1000 + nState_SEQ_Enabling;
		END_IF		
		
		
	150: // Enable group
		hr :=THIS^.ipGroup.Enable();
		
		IF CheckOk(hr) THEN 
			nState_SEQ_Enabling := 160;
		ELSE
			nState_SEQ_Enabling := 1000 + nState_SEQ_Enabling;
		END_IF	
		
		
	160: // Enabling group
		hr := THIS^.ipGroup.HR;
		
		IF THIS^.ipGroup.GroupEnabled THEN 
			nState_SEQ_Enabling := 999;
		ELSIF FAILED(hr) THEN
			nState_SEQ_Enabling := 1000 + nState_SEQ_Enabling;
		END_IF	
		
		
	999: // Done
		Enabling := S_OK;

		
	1000..1999://Error
		hr := GetMostSignificant(hrLastCycle, E_FAIL);
	
END_CASE


//Timeout after to long stay in one of the following seq.
fbTimeOutSeq.IN := (nState_SEQ_Enabling = 2) OR (nState_SEQ_Enabling = 5);
fbTimeOutSeq.PT := T#5S;
fbTimeOutSeq();

IF fbTimeOutSeq.Q THEN
	//next seq is error
	nState_SEQ_Enabling := 1000 + nState_SEQ_Enabling;
END_IF

//store last information
hrLastCycle := hr;

// Propagate error
IF FAILED(hr) THEN
	Enabling := hr;
END_IF
END_METHOD

METHOD Initialize : HRESULT
VAR
	hr : HRESULT;
END_VAR

VAR
	fbStationsToCheck : CHALET_BaseComponents.FB_CH_List;
	ipStationToCheck, ipTempStation : I_XTS_Station;
END_VAR
VAR_INST
	//This error cannot be reset. Requires a reset cold
	{attribute 'hide'}	
	fbInitError : FB_TcAlarm;
END_VAR
//Check Error during FB_Init
IF THIS^.bErrorDuringFbInit THEN
	IF NOT fbInitError.bRaised THEN 
		//This error cannot be reset. Requires a reset cold
		fbInitError.CreateEx(stEventEntry:=TC_EVENTS.CHALET_XTS_Events.ErrorFBinit, ipSourceInfo := THIS^.fbSourceInfo, bWithConfirmation := FALSE);
		fbInitError.Raise(0);
	END_IF
	Initialize:= E_FAIL;
	RETURN;
END_IF	

//Check if Envirement and Group is existing
IF THIS^.ipEnvironment = 0 OR THIS^.ipGroup = 0 THEN
	IF NOT fbInitError.bRaised THEN 
		//This error cannot be reset. Requires a reset cold
		fbInitError.CreateEx(stEventEntry:=TC_EVENTS.CHALET_XTS_Events.InitializationInvalideParameter, ipSourceInfo := THIS^.fbSourceInfo, bWithConfirmation := FALSE);
		fbInitError.Raise(0);
	END_IF
	Initialize:= E_FAIL;
	RETURN;
END_IF	


//Check for stations on the same position
fbStationsToCheck.Duplicate(THIS^.fbStations);
// go through the list and search the station in front
fbStationsToCheck.ResetIterator();
WHILE fbStationsToCheck.HasNextObject() DO
	IF ToStation(fbStationsToCheck.GetNextObject(), ipStationToCheck) THEN
		fbStations.ResetIterator();
		WHILE THIS^.fbStations.HasNextObject() DO
			IF ToStation(THIS^.fbStations.GetNextObject(), ipTempStation) THEN
				// Error - Same LUID(Name) of 2 stations
				IF (ipStationToCheck.LUID = ipTempStation.LUID) AND (ipStationToCheck <> ipTempStation) THEN
					IF NOT fbInitError.bRaised THEN 
						//This error cannot be reset. Requires a reset cold
						fbInitError.CreateEx(stEventEntry:=TC_EVENTS.CHALET_XTS_Events.DublicateStationNames, ipSourceInfo := THIS^.fbSourceInfo, bWithConfirmation := FALSE);
						fbInitError.ipArguments.AddStringByValue(ipTempStation.LUID);
						fbInitError.Raise(0);
					END_IF
					Initialize:= E_FAIL;
					RETURN;	
				END_IF
				// Error - Same Position of 2 stations
				IF (ipStationToCheck.PositionOnTrack = ipTempStation.PositionOnTrack) AND (ipStationToCheck <> ipTempStation) THEN
					IF NOT fbInitError.bRaised THEN 
						//This error cannot be reset. Requires a reset cold
						fbInitError.CreateEx(stEventEntry:=TC_EVENTS.CHALET_XTS_Events.DublicateStationPositions, ipSourceInfo := THIS^.fbSourceInfo, bWithConfirmation := FALSE);
						fbInitError.ipArguments.AddStringByValue(ipTempStation.LUID).AddStringByValue(ipStationToCheck.LUID);
						fbInitError.Raise(0);
					END_IF
					Initialize:= E_FAIL;
					RETURN;	
				END_IF
			END_IF
		END_WHILE
	END_IF
END_WHILE


hr := GetMostSignificant(hr, ipEnvironment.Initialize());	
//Init envirement first to get access to XTS_Utility
IF THIS^.ipEnvironment.UtilityEnvirement.P_IsInitialized THEN
	hr := GetMostSignificant(hr, fbMovers.Initialize());	
	hr := GetMostSignificant(hr, ipGroup.Initialize());	
	hr := GetMostSignificant(hr, fbStations.Initialize());	
	hr := GetMostSignificant(hr, fbZones.Initialize());	
	hr := GetMostSignificant(hr, fbTriggers.Initialize());	
ELSE
	hr := GetMostSignificant(hr, S_PENDING);
END_IF	


THIS^.bInitDone := (hr = S_OK);
Initialize:= hr;
END_METHOD

{attribute 'monitoring':='call'}
PROPERTY Initialized : BOOL
GET
Initialized := bInitDone;
END_GET
END_PROPERTY

METHOD LinkEnvironment : HRESULT
VAR_INPUT
	ipEnvironment	: CHALET_BaseComponents.I_CH_Object;
END_VAR

VAR
	ipXtsEnvironment : I_Xts_Environment;
END_VAR
IF ipEnvironment <> 0 AND_THEN __QUERYINTERFACE(ipEnvironment, ipXtsEnvironment) THEN
	THIS^.ipEnvironment := ipXtsEnvironment;
	LinkEnvironment := S_OK;
ELSE
	LinkEnvironment := E_FAIL;
	THIS^.bErrorDuringFbInit := TRUE;
END_IF
END_METHOD

METHOD LinkGroup : HRESULT
VAR_INPUT
	ipGroup	: CHALET_BaseComponents.I_CH_Object;
END_VAR

VAR
	ipXtsGroup : I_XTS_Group;
END_VAR
IF ipGroup <> 0 AND_THEN __QUERYINTERFACE(ipGroup, ipXtsGroup) THEN
	THIS^.ipGroup := ipXtsGroup;
	LinkGroup := S_OK;
ELSE
	LinkGroup := E_FAIL;
	THIS^.bErrorDuringFbInit := TRUE;
END_IF
END_METHOD

METHOD RegisterMover : HRESULT
VAR_INPUT
	ipMover	: CHALET_BaseComponents.I_CH_Object;
END_VAR

VAR
	ipXtsMover : I_XTS_Mover;
END_VAR
IF ipMover = 0 THEN
	//Invalide interface	
	THIS^.bErrorDuringFbInit := TRUE;
	RegisterMover := E_FAIL;
	
ELSIF NOT __QUERYINTERFACE(ipMover, ipXtsMover) THEN
	//The required interface is missing
	THIS^.bErrorDuringFbInit := TRUE;
	RegisterMover := E_FAIL;
	
ELSIF THIS^.fbMovers.IsFull THEN
	//List is full
	THIS^.bErrorDuringFbInit := TRUE;
	RegisterMover := E_FAIL;
	
ELSIF THIS^.bInitDone THEN
	//To late. System is initilized
	THIS^.bErrorDuringFbInit := TRUE;
	RegisterMover := E_FAIL;
	
ELSE
	
	THIS^.fbMovers.AddObject(ipMover);
END_IF
END_METHOD

METHOD RegisterStation : HRESULT
VAR_INPUT
	ipStation	: CHALET_BaseComponents.I_CH_Object;
END_VAR

VAR
	ipXtsStation : I_XTS_Station;
END_VAR
IF ipStation = 0 THEN
	//Invalide interface	
	THIS^.bErrorDuringFbInit := TRUE;
	RegisterStation := E_FAIL;
	
ELSIF NOT __QUERYINTERFACE(ipStation, ipXtsStation) THEN
	//The required interface is missing
	THIS^.bErrorDuringFbInit := TRUE;
	RegisterStation := E_FAIL;
	
ELSIF THIS^.fbStations.IsFull THEN
	//List is full
	THIS^.bErrorDuringFbInit := TRUE;
	RegisterStation := E_FAIL;
	
ELSIF THIS^.bInitDone THEN
	//To late. System is initilized
	THIS^.bErrorDuringFbInit := TRUE;
	RegisterStation := E_FAIL;
		
ELSE
	
	THIS^.fbStations.AddObject(ipStation);
END_IF
END_METHOD

METHOD RegisterTrigger : HRESULT
VAR_INPUT
	ipTrigger	: CHALET_BaseComponents.I_CH_Object;
END_VAR
VAR
	ipXtsTrigger : I_XTS_Trigger;
END_VAR
IF ipTrigger = 0 THEN
	//Invalide interface	
	THIS^.bErrorDuringFbInit := TRUE;
	RegisterTrigger := E_FAIL;
	
ELSIF NOT __QUERYINTERFACE(ipTrigger, ipXtsTrigger) THEN
	//The required interface is missing
	THIS^.bErrorDuringFbInit := TRUE;
	RegisterTrigger := E_FAIL;
	
ELSIF THIS^.fbTriggers.IsFull THEN
	//List is full
	THIS^.bErrorDuringFbInit := TRUE;
	RegisterTrigger := E_FAIL;
	
ELSIF THIS^.bInitDone THEN
	//To late. System is initilized
	THIS^.bErrorDuringFbInit := TRUE;
	RegisterTrigger := E_FAIL;
		
ELSE
	
	THIS^.fbTriggers.AddObject(ipTrigger);
END_IF
END_METHOD

METHOD RegisterZone : HRESULT
VAR_INPUT
	ipZone	: CHALET_BaseComponents.I_CH_Object;
END_VAR
VAR
	ipXtsZone : I_XTS_Zone;
END_VAR
IF ipZone = 0 THEN
	//Invalide interface	
	THIS^.bErrorDuringFbInit := TRUE;
	RegisterZone := E_FAIL;

ELSIF NOT __QUERYINTERFACE(ipZone, ipXtsZone) THEN
	//The required interface is missing
	THIS^.bErrorDuringFbInit := TRUE;
	RegisterZone := E_FAIL;
	
ELSIF THIS^.fbZones.IsFull THEN
	//List is full
	THIS^.bErrorDuringFbInit := TRUE;
	RegisterZone := E_FAIL;
	
ELSIF THIS^.bInitDone THEN
	//To late. System is initilized
	THIS^.bErrorDuringFbInit := TRUE;
	RegisterZone := E_FAIL;
		
ELSE
	
	THIS^.fbZones.AddObject(ipZone);	
END_IF
END_METHOD

{attribute 'monitoring':='call'}
PROPERTY Environment : I_XTS_Environment
GET
Environment := THIS^.ipEnvironment;
END_GET
END_PROPERTY

{attribute 'monitoring':='call'}
PROPERTY Feedback : CHALET_BaseComponents.I_CH_Feedback
GET
Feedback := THIS^.fbFeedback;
END_GET
END_PROPERTY

METHOD getMoverInFront : I_Xts_Mover
VAR_INPUT
	ipMover	: I_Xts_Mover;
END_VAR

VAR
	fPosOnTrack			: LREAL;
	ipTempMover 		: I_XTS_Mover;
	fTempPosOnTrack		: LREAL;
	fTempDistBetween 	: LREAL;
	
	fFoundDistBetween : LREAL := CHALET_BaseComponents.GVL_Datatypes.cMaxLreal;
	ipFoundMover	: I_Xts_Mover;
END_VAR
//use NcToPlc.ModuloActPos because iMover.PositionOnTrack is not ready during init
//get an copy of the mover list 
//fbTempListOfMovers.Duplicate(THIS^.fbMovers);


// get postion of myself
fPosOnTrack := ipMover.getAxisRef.NcToPlc.ModuloActPos;

// go through the list and search the mover in front
THIS^.fbMovers.ResetIterator();
WHILE THIS^.fbMovers.HasNextObject() DO
	IF ToMover(THIS^.fbMovers.GetNextObject(), ipTempMover) THEN
		// if Mover is myself, skipp
		IF ipTempMover <> ipMover THEN
			// calc distance to Mover in positive direction
			fTempDistBetween := FUN_GetDistToPosModulo(fActualPosition := fPosOnTrack, fTargedPosition := ipTempMover.getAxisRef.NcToPlc.ModuloActPos, fModulo := TrackLength);
	
	
			// check if Mover is closer then last one
			IF fFoundDistBetween > fTempDistBetween THEN 
				fFoundDistBetween := fTempDistBetween;
				ipFoundMover := ipTempMover;
			END_IF
		END_IF
	END_IF
END_WHILE

getMoverInFront := ipFoundMover;
END_METHOD

METHOD getStationInFront : I_XTS_Station
VAR_INPUT
	ipStation	: I_XTS_Station;
END_VAR
VAR
	fPosOnTrack			: LREAL;
	
	ipTempStation 		: I_XTS_Station;
	fTempPosOnTrack		: LREAL;
	fTempDistBetween 	: LREAL;
	
	fFoundDistBetween 	: LREAL := CHALET_BaseComponents.GVL_Datatypes.cMaxLreal;
	ipFoundStation		: I_XTS_Station;
END_VAR
// get postion of myself
fPosOnTrack := ipStation.PositionOnTrack;

// go through the list and search the station in front
THIS^.fbStations.ResetIterator();
WHILE THIS^.fbStations.HasNextObject() DO
	IF ToStation(THIS^.fbStations.GetNextObject(), ipTempStation) THEN
		// calc distance to Station
		fTempDistBetween := ipTempStation.PositionOnTrack - fPosOnTrack;		
		
		// if Station is behinde me or it is myself -> add Modulo
		IF fTempDistBetween <= 0 THEN 
			fTempDistBetween := fTempDistBetween + TrackLength;			
		END_IF

		// check if Station is closer then last one
		IF fFoundDistBetween > fTempDistBetween THEN 
			fFoundDistBetween := fTempDistBetween;
			ipFoundStation := ipTempStation;
		END_IF
		
	END_IF
END_WHILE

getStationInFront := ipFoundStation;
END_METHOD

{attribute 'monitoring':='call'}
PROPERTY Movers : CHALET_BaseComponents.I_CH_LIST
GET
Movers := THIS^.fbMovers;
END_GET
END_PROPERTY

METHOD Reset : HRESULT
VAR
	hr : HRESULT;
	bOk : BOOL := TRUE;
	ipTempMover : I_XTS_Mover;
END_VAR
// Reset movers
THIS^.fbMovers.ResetIterator();
WHILE THIS^.fbMovers.HasNextObject() DO
	IF ToMover(THIS^.fbMovers.GetNextObject(),ipTempMover) THEN
		hr := GetMostSignificant(hr, ipTempMover.Reset());
	END_IF
END_WHILE
	
// Reset groupe	
IF THIS^.ipGroup <> 0 THEN
	GetMostSignificant(hr, THIS^.ipGroup.Reset());
END_IF

Reset := hr;
END_METHOD

METHOD Station : I_XTS_Station_PLC
VAR_INPUT
	sLUID	: STRING;
END_VAR
//IF no station was found, INTERFACE is 0 -> can generate fatal error
__QUERYINTERFACE(THIS^.fbStations.FindLUID(sLUID),Station);
END_METHOD

{attribute 'monitoring':='call'}
PROPERTY Stations : CHALET_BaseComponents.I_CH_LIST
GET
Stations := THIS^.fbStations;
END_GET
END_PROPERTY

PROPERTY SuppressAllDynamicsChanges : BOOL
SET
VAR
	ipTempStationPlc : I_XTS_Station_PLC;
END_VAR
// go through the list and write request to it
THIS^.fbStations.ResetIterator();
WHILE THIS^.fbStations.HasNextObject() DO
	IF ToStation_PLC(THIS^.fbStations.GetNextObject(), ipTempStationPlc) THEN
		ipTempStationPlc.SuppressDynamicsChange := SuppressAllDynamicsChanges;
	END_IF
END_WHILE
END_SET
END_PROPERTY

{attribute 'monitoring':='call'}
PROPERTY TrackLength : LREAL
GET
TrackLength := THIS^.ipEnvironment.TrackLength;
END_GET
END_PROPERTY

{attribute 'monitoring':='call'}
PROPERTY Triggers : CHALET_BaseComponents.I_CH_LIST
GET
Triggers := THIS^.fbTriggers;
END_GET
END_PROPERTY

METHOD Update : HRESULT
VAR_INPUT
END_VAR
VAR
	hr : HRESULT;
END_VAR
//Force to do an init at beginn
IF NOT THIS^.Initialized THEN
	THIS^.Initialize();
	RETURN;
END_IF

hr := S_OK;

hr := GetMostSignificant(hr, THIS^.Enabling());	
hr := GetMostSignificant(hr, THIS^.Disabling());	

THIS^.fbFeedback.HR := hr;

hr := GetMostSignificant(hr, THIS^.fbMovers.Update());	
hr := GetMostSignificant(hr, THIS^.fbStations.Update());	
hr := GetMostSignificant(hr, THIS^.fbZones.Update());	
hr := GetMostSignificant(hr, THIS^.fbTriggers.Update());	

//zzz Todo vllt könnte hier das CH_Object verwendet werden
hr := GetMostSignificant(hr, THIS^.ipGroup.Update());	
hr := GetMostSignificant(hr, THIS^.ipEnvironment.Update());	

Update:= hr;
END_METHOD

{attribute 'monitoring':='call'}
PROPERTY Zones : CHALET_BaseComponents.I_CH_LIST
GET
Zones := THIS^.fbZones;
END_GET
END_PROPERTY

END_FUNCTION_BLOCK

// COMPENENTs/System/I_XTS_System_PLC
INTERFACE I_XTS_System_PLC

METHOD Disable : I_CH_Feedback
VAR_INPUT
END_VAR
END_METHOD

{attribute 'monitoring':='call'}
PROPERTY Disabled : Bool
GET
END_GET
END_PROPERTY

METHOD Enable : I_CH_Feedback
VAR_INPUT
END_VAR
END_METHOD

{attribute 'monitoring':='call'}
PROPERTY Enabled : Bool
GET
END_GET
END_PROPERTY

{attribute 'monitoring':='call'}
PROPERTY Feedback : CHALET_BaseComponents.I_CH_Feedback
GET
END_GET
END_PROPERTY

METHOD Initialize : HRESULT
VAR_INPUT
END_VAR
END_METHOD

{attribute 'monitoring':='call'}
PROPERTY Initialized : BOOL
GET
END_GET
END_PROPERTY

METHOD Reset : HRESULT
VAR_INPUT
END_VAR
END_METHOD

METHOD Station : I_XTS_Station_PLC
VAR_INPUT
	sLUID : STRING;
END_VAR
END_METHOD

PROPERTY SuppressAllDynamicsChanges : BOOL
SET
END_SET
END_PROPERTY

{attribute 'monitoring':='call'}
PROPERTY TrackLength : LREAL
GET
END_GET
END_PROPERTY

METHOD Update : HRESULT
VAR_INPUT
END_VAR
END_METHOD

END_INTERFACE
